// TIA Portal V16 export
// export: Created 2025-11-10T21:24:54.1591457Z, ExportSetting WithDefaults, DisplayName Totally Integrated Automation Portal, DisplayVersion V16, DisplayName TIA Portal Version Control Interface, DisplayVersion V16, DisplayName TIA Portal Openness, DisplayVersion V16, DisplayName STEP 7 Professional, DisplayVersion V16, DisplayName STEP 7 Safety, DisplayVersion V16, DisplayName WinCC Advanced, DisplayVersion V16
ORGANIZATION_BLOCK "OB1"   // OB1, LAD, ProgramCycle
TITLE = MAIN Program - Sweep
VERSION : 0.1
// MAIN Program Block (Release)
// stored: IsIECCheckEnabled false
   VAR_TEMP
      Temp_0 : Byte;
      Temp_1 : Byte;
      Temp_2 : Byte;
      Temp_3 : Byte;
      Temp_4 : Byte;
      Temp_5 : Byte;
      Temp_6 : Int;
      Temp_7 : Int;
      Temp_8 : Int;
      Temp_9 : Date_And_Time;
      Temp_10 : DWord;
      EncoderDirection : Bool;
      HomingActive : Bool;
      EncError : Bool;
      SafetyActive : Bool;
      "Spare Drive 6" : Bool;
      "Spare Drive 7" : Bool;
      "Spare Drive 8" : Bool;
      "Spare Drive 9" : Bool;
      "Spare Drive 10" : Bool;
      SAFE_OK_Signal : Bool;
      Raw_Position : Real;
      Encoder : Int;
      Gate : Bool;
      GATESTP : Bool;
      OTERRA : Bool;
      Direct : Bool;
      Prepar : Bool;
      CMPV1 : Bool;
      CMPV2 : Bool;
      RESSYNC : Bool;
      RESZERO : Bool;
      OTERR : Bool;
      UnscPos : Int;
      Sc_Pos : Int;
      ActEncPos : Real;
      Start_ReferenceRun : Bool;
      ReferenceSwitch_Input : Bool;
      "Reference Position" : Real;
      "Jog FWD" : Bool;
      "Jog REV" : Bool;
      RefSwitchTemp : Bool;
      RefPosDint : DInt;
      RefPosInt : Real;
      Start_Movement : Bool;
      ClockTime : Int;
      LT_Time : Date_And_Time;
      Summer : Bool;
      SystemStartUp : Bool;
      StartupLow : Bool;
      ManualSensorOverride : Bool;
      Axis1_ScaledPosition : Real;
      Axis1_ActualEncPosition : Real;
      ActivateProductBufferV2 : Bool;
      ActivateProductBufferV3 : Bool;
      SetZPulse : Bool;
      Enc2_AboveZero : DInt;
      MinValue : DInt;
      EncBelowZero : Bool;
      SafeEncValue : Real;
      Enc2_Real : Real;
      ScPos : Real;
      UseOldDriveManager : Bool;
      NotUsed : Bool;
      Door2 : Bool;
      Resettt : Bool;
      BlkMovReturn : Int;
      BlkMovReturn2 : Int;
      ServoAxis3RefRun : Bool;
   END_VAR
   VAR_TEMP   // added for the SCL form of the ladder/FBD networks
      _w1 : Bool;
   END_VAR
BEGIN

REGION Network 1: System Startup
   // Network for detecting System Start-up.
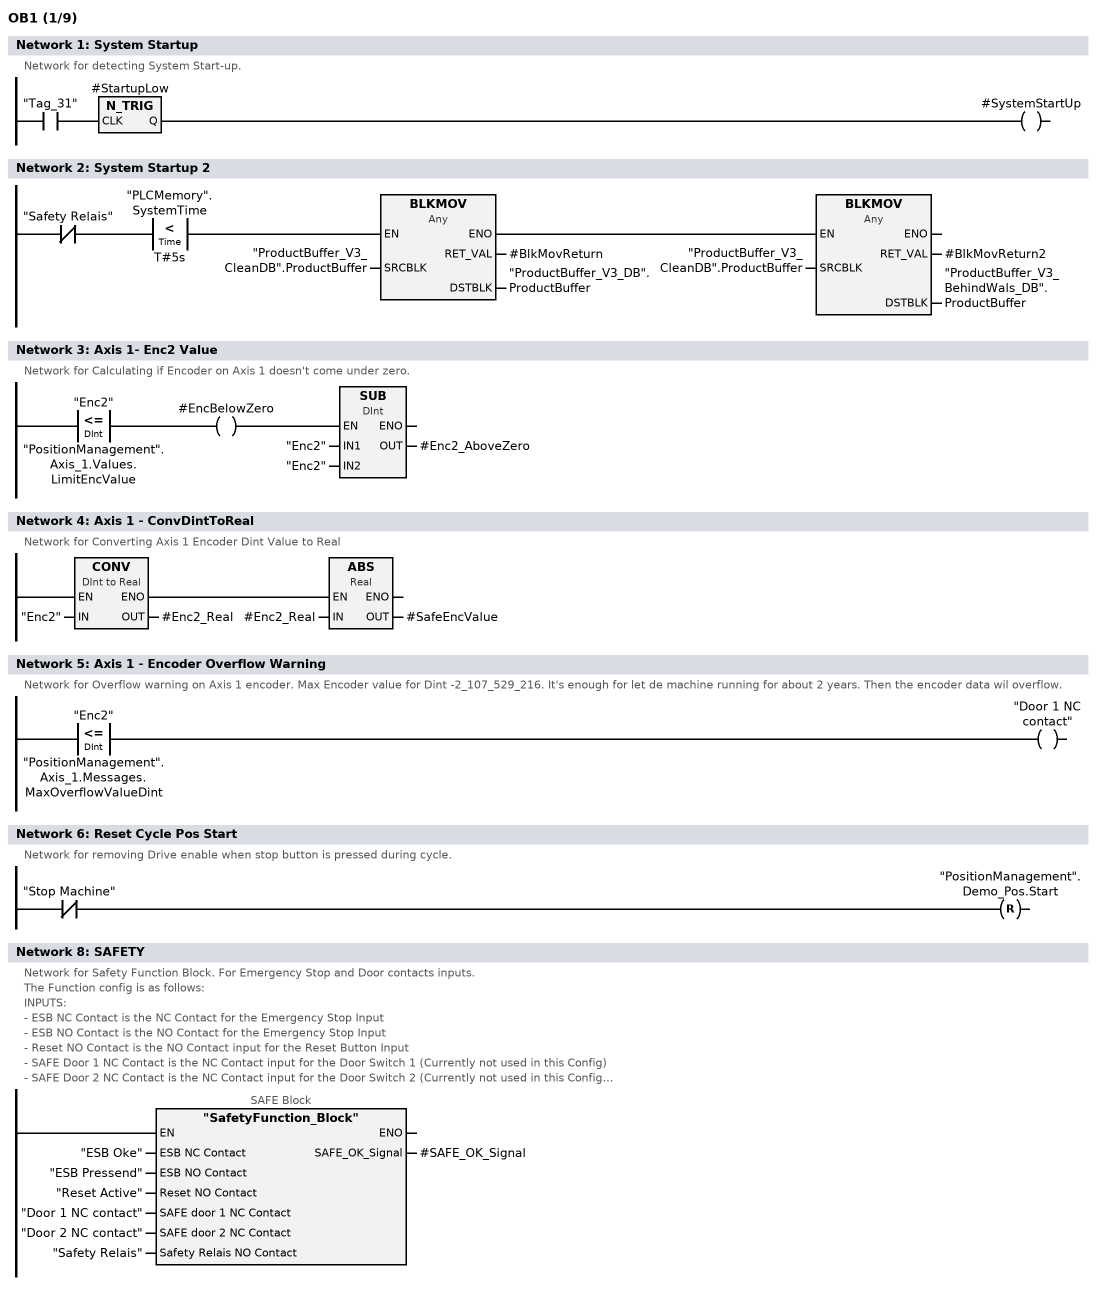
   RUNG wire#powerrail
      Contact( "Tag_31" )
      N_Trig( #StartupLow )
      Coil( #SystemStartUp )
   END_RUNG
   // the same network as SCL:
   #_w1 := NOT "Tag_31" AND #StartupLow;   // falling edge
   #StartupLow := "Tag_31";
   #SystemStartUp := #_w1;
END_REGION

REGION Network 2: System Startup 2
   RUNG wire#powerrail
      I_Contact( "Safety Relais" )
      { S7_Templates := "SrcType := Time" } LT_Contact(in1 := "PLCMemory".SystemTime, in2 := T#5s)
      { S7_Templates := "blk_type := Any" } BLKMOV(SRCBLK := "ProductBuffer_V3_CleanDB".ProductBuffer, RET_VAL => #BlkMovReturn, DSTBLK => "ProductBuffer_V3_DB".ProductBuffer)
      { S7_Templates := "blk_type := Any" } BLKMOV(SRCBLK := "ProductBuffer_V3_CleanDB".ProductBuffer, RET_VAL => #BlkMovReturn2, DSTBLK => "ProductBuffer_V3_BehindWals_DB".ProductBuffer)
   END_RUNG
   // the same network as SCL:
   #BlkMovReturn := BLKMOV(EN := NOT "Safety Relais" AND ("PLCMemory".SystemTime < T#5s),
                           SRCBLK := "ProductBuffer_V3_CleanDB".ProductBuffer,
                           DSTBLK => "ProductBuffer_V3_DB".ProductBuffer,
                           ENO => #_w1);
   IF #_w1 THEN
       #BlkMovReturn2 := BLKMOV(SRCBLK := "ProductBuffer_V3_CleanDB".ProductBuffer,
                               DSTBLK => "ProductBuffer_V3_BehindWals_DB".ProductBuffer);
   END_IF;
END_REGION

REGION Network 3: Axis 1- Enc2 Value
   // Network for Calculating if Encoder on Axis 1 doesn't come under zero.
   RUNG wire#powerrail
      { S7_Templates := "SrcType := DInt" } LE_Contact(in1 := "Enc2", in2 := "PositionManagement".Axis_1.Values.LimitEncValue)
      Coil( #EncBelowZero )
      { S7_Templates := "SrcType := DInt"; S7_GenerateENO := "TRUE" } Sub(in1 := "Enc2", in2 := "Enc2", out => #Enc2_AboveZero)
   END_RUNG
   // the same network as SCL:
   #EncBelowZero := "Enc2" <= "PositionManagement".Axis_1.Values.LimitEncValue;
   IF #EncBelowZero THEN #Enc2_AboveZero := "Enc2" - "Enc2"; END_IF;
END_REGION

REGION Network 4: Axis 1 - ConvDintToReal
   // Network for Converting Axis 1 Encoder Dint Value to Real
   RUNG wire#powerrail
      { S7_Templates := "[SrcType := DInt, DestType := Real]"; S7_GenerateENO := "TRUE" } Convert(in := "Enc2", out => #Enc2_Real)
      { S7_Templates := "SrcType := Real"; S7_GenerateENO := "TRUE" } Abs(in := #Enc2_Real, out => #SafeEncValue)
   END_RUNG
   // the same network as SCL:
   // ENO of a box is taken as its EN; it also drops when the box reports an error
   #Enc2_Real := DINT_TO_REAL("Enc2");
   #SafeEncValue := ABS(#Enc2_Real);
END_REGION

REGION Network 5: Axis 1 - Encoder Overflow Warning
   // Network for Overflow warning on Axis 1 encoder. Max Encoder value for Dint -2_107_529_216. It's enough for let de machine running for about 2 years. Then the encoder data wil overflow.
   RUNG wire#powerrail
      { S7_Templates := "SrcType := DInt" } LE_Contact(in1 := "Enc2", in2 := "PositionManagement".Axis_1.Messages.MaxOverflowValueDint)
      Coil( "Door 1 NC contact" )
   END_RUNG
   // the same network as SCL:
   "Door 1 NC contact" := "Enc2" <= "PositionManagement".Axis_1.Messages.MaxOverflowValueDint;
END_REGION

REGION Network 6: Reset Cycle Pos Start
   // Network for removing Drive enable when stop button is pressed during cycle.
   RUNG wire#powerrail
      I_Contact( "Stop Machine" )
      R_Coil( "PositionManagement".Demo_Pos.Start )
   END_RUNG
   // the same network as SCL:
   IF NOT "Stop Machine" THEN "PositionManagement".Demo_Pos.Start := FALSE; END_IF;
END_REGION

REGION Network 7: Retain Veriables (Not Used)
   // Spare Network Currently not used
END_REGION

REGION Network 8: SAFETY
   // Network for Safety Function Block. For Emergency Stop and Door contacts inputs.
   // The Function config is as follows:
   // 
   // INPUTS:
   // - ESB NC Contact is the NC Contact for the Emergency Stop Input
   // - ESB NO Contact is the NO Contact for the Emergency Stop Input
   // - Reset NO Contact is the NO Contact input for the Reset Button Input
   // - SAFE Door 1 NC Contact is the NC Contact input for the Door Switch 1 (Currently not used in this Config)
   // - SAFE Door 2 NC Contact is the NC Contact input for the Door Switch 2 (Currently not used in this Config)
   // - Safety Relais NO Contact is the NO Contact Input for feedback whenether the Safety Relais is powered or not.
   // 
   // OUTPUTS:
   // - SAFE_OK_Signal is the output for the SAFE OK signal, it's HIGH when all safety inputs are HIGH, en when Reset is given.
   RUNG wire#powerrail
      "SafetyFunction_Block"("ESB NC Contact" := "ESB Oke", "ESB NO Contact" := "ESB Pressend", "Reset NO Contact" := "Reset Active", "SAFE door 1 NC Contact" := "Door 1 NC contact", "SAFE door 2 NC Contact" := "Door 2 NC contact", "Safety Relais NO Contact" := "Safety Relais", SAFE_OK_Signal => #SAFE_OK_Signal)   // SAFE Block
   END_RUNG
   // the same network as SCL:
   "SafetyFunction_Block"("ESB NC Contact" := "ESB Oke",   // SAFE Block
                          "ESB NO Contact" := "ESB Pressend",
                          "Reset NO Contact" := "Reset Active",
                          "SAFE door 1 NC Contact" := "Door 1 NC contact",
                          "SAFE door 2 NC Contact" := "Door 2 NC contact",
                          "Safety Relais NO Contact" := "Safety Relais",
                          SAFE_OK_Signal => #SAFE_OK_Signal);
END_REGION

REGION Network 9: SAFE Signal
   // Network for internal SAFETY OK Confirmation
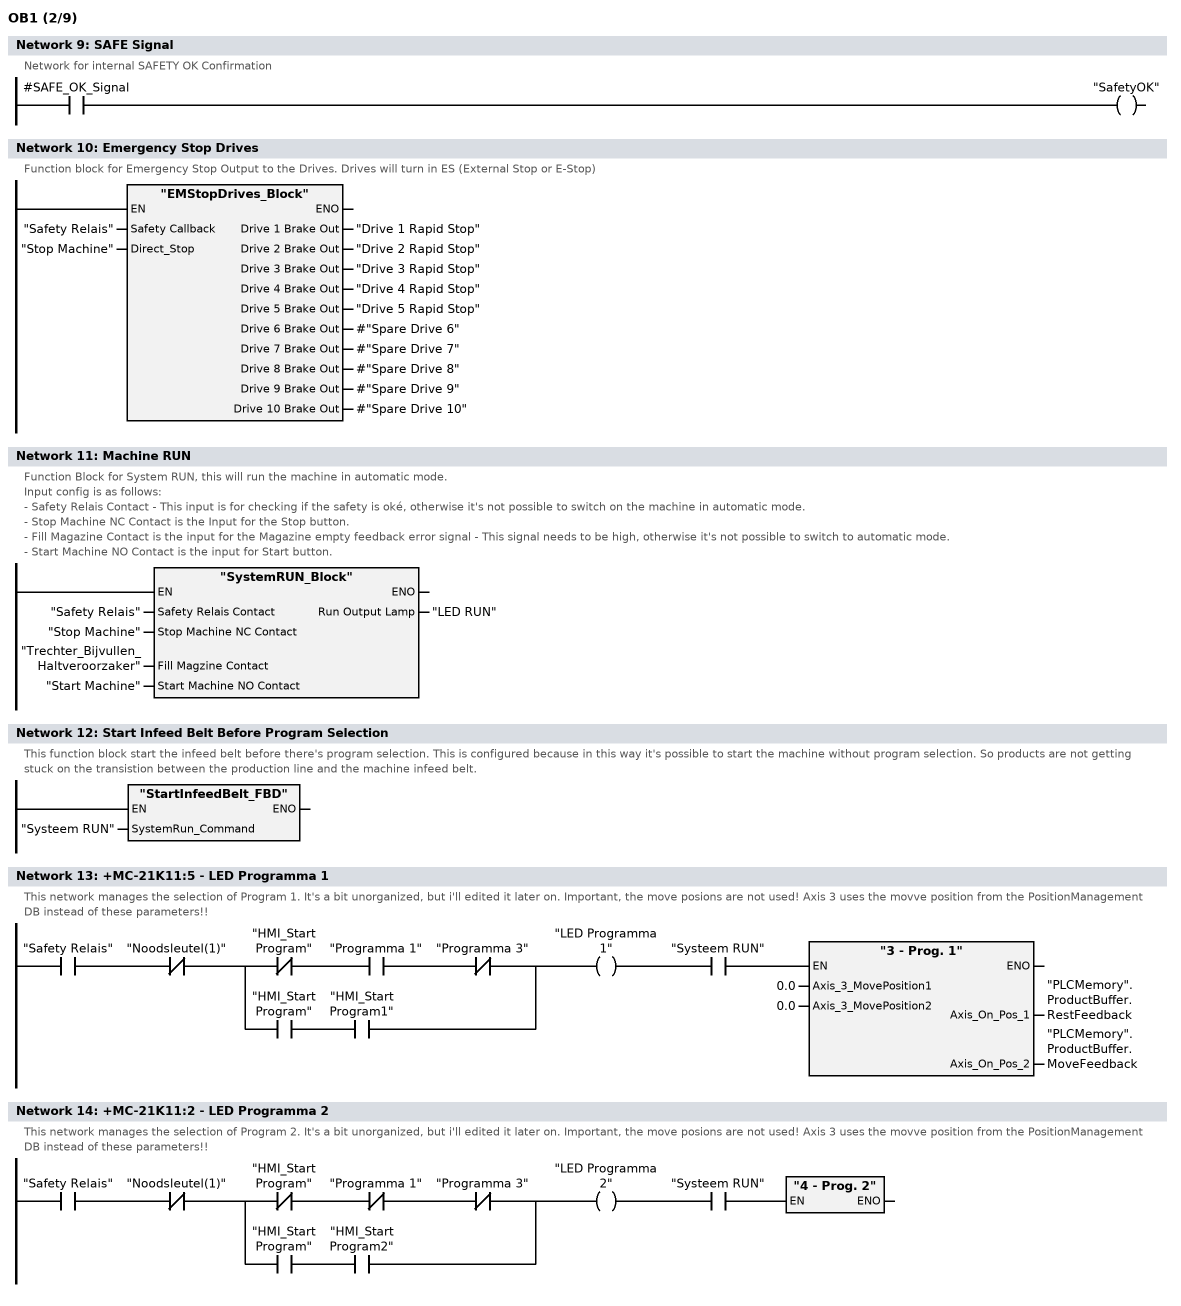
   RUNG wire#powerrail
      Contact( #SAFE_OK_Signal )
      Coil( "SafetyOK" )
   END_RUNG
   // the same network as SCL:
   "SafetyOK" := #SAFE_OK_Signal;
END_REGION

REGION Network 10: Emergency Stop Drives
   // Function block for Emergency Stop Output to the Drives. Drives will turn in ES (External Stop or E-Stop)
   RUNG wire#powerrail
      "EMStopDrives_Block"("Safety Callback" := "Safety Relais", Direct_Stop := "Stop Machine", "Drive 1 Brake Out" => "Drive 1 Rapid Stop", "Drive 2 Brake Out" => "Drive 2 Rapid Stop", "Drive 3 Brake Out" => "Drive 3 Rapid Stop", "Drive 4 Brake Out" => "Drive 4 Rapid Stop", "Drive 5 Brake Out" => "Drive 5 Rapid Stop", "Drive 6 Brake Out" => #"Spare Drive 6", "Drive 7 Brake Out" => #"Spare Drive 7", "Drive 8 Brake Out" => #"Spare Drive 8", "Drive 9 Brake Out" => #"Spare Drive 9", "Drive 10 Brake Out" => #"Spare Drive 10")
   END_RUNG
   // the same network as SCL:
   "EMStopDrives_Block"("Safety Callback" := "Safety Relais",
                        Direct_Stop := "Stop Machine",
                        "Drive 1 Brake Out" => "Drive 1 Rapid Stop",
                        "Drive 2 Brake Out" => "Drive 2 Rapid Stop",
                        "Drive 3 Brake Out" => "Drive 3 Rapid Stop",
                        "Drive 4 Brake Out" => "Drive 4 Rapid Stop",
                        "Drive 5 Brake Out" => "Drive 5 Rapid Stop",
                        "Drive 6 Brake Out" => #"Spare Drive 6",
                        "Drive 7 Brake Out" => #"Spare Drive 7",
                        "Drive 8 Brake Out" => #"Spare Drive 8",
                        "Drive 9 Brake Out" => #"Spare Drive 9",
                        "Drive 10 Brake Out" => #"Spare Drive 10");
END_REGION

REGION Network 11: Machine RUN
   // Function Block for System RUN, this will run the machine in automatic mode.
   // Input config is as follows:
   // - Safety Relais Contact - This input is for checking if the safety is oké, otherwise it's not possible to switch on the machine in automatic mode.
   // - Stop Machine NC Contact is the Input for the Stop button.
   // - Fill Magazine Contact is the input for the Magazine empty feedback error signal - This signal needs to be high, otherwise it's not possible to switch to automatic mode.
   // - Start Machine NO Contact is the input for Start button.
   RUNG wire#powerrail
      "SystemRUN_Block"("Safety Relais Contact" := "Safety Relais", "Stop Machine NC Contact" := "Stop Machine", "Fill Magzine Contact" := "Trechter_Bijvullen_Haltveroorzaker", "Start Machine NO Contact" := "Start Machine", "Run Output Lamp" => "LED RUN")
   END_RUNG
   // the same network as SCL:
   "SystemRUN_Block"("Safety Relais Contact" := "Safety Relais",
                     "Stop Machine NC Contact" := "Stop Machine",
                     "Fill Magzine Contact" := "Trechter_Bijvullen_Haltveroorzaker",
                     "Start Machine NO Contact" := "Start Machine",
                     "Run Output Lamp" => "LED RUN");
END_REGION

REGION Network 12: Start Infeed Belt Before Program Selection
   // This function block start the infeed belt before there's program selection. This is configured because in this way it's possible to start the machine without program selection. So products are not getting stuck on the transistion between the production line and the machine infeed belt.
   RUNG wire#powerrail
      "StartInfeedBelt_FBD"(SystemRun_Command := "Systeem RUN")
   END_RUNG
   // the same network as SCL:
   "StartInfeedBelt_FBD"(SystemRun_Command := "Systeem RUN");
END_REGION

REGION Network 13: +MC-21K11:5 - LED Programma 1
   // This network manages the selection of Program 1. It's a bit unorganized, but i'll edited it later on. Important, the move posions are not used! Axis 3 uses the movve position from the PositionManagement DB instead of these parameters!!
   RUNG wire#powerrail
      Contact( "Safety Relais" )
      I_Contact( "Noodsleutel(1)" )
      wire#w1
      I_Contact( "HMI_StartProgram" )
      Contact( "Programma 1" )
      I_Contact( "Programma 3" )
      wire#w2
      Coil( "LED Programma 1" )
      Contact( "Systeem RUN" )
      "3 - Prog. 1"(Axis_3_MovePosition1 := 0.0, Axis_3_MovePosition2 := 0.0, Axis_On_Pos_1 => "PLCMemory".ProductBuffer.RestFeedback, Axis_On_Pos_2 => "PLCMemory".ProductBuffer.MoveFeedback)
   END_RUNG
   RUNG wire#w1
      Contact( "HMI_StartProgram" )
      Contact( "HMI_StartProgram1" )
   END_RUNG wire#w2
   // the same network as SCL:
   "LED Programma 1" := "Safety Relais" AND NOT "Noodsleutel(1)" AND ((NOT "HMI_StartProgram" AND "Programma 1" AND NOT "Programma 3") OR ("HMI_StartProgram" AND "HMI_StartProgram1"));
   IF "LED Programma 1" AND "Systeem RUN" THEN
       "3 - Prog. 1"(Axis_3_MovePosition1 := 0.0,
                     Axis_3_MovePosition2 := 0.0,
                     Axis_On_Pos_1 => "PLCMemory".ProductBuffer.RestFeedback,
                     Axis_On_Pos_2 => "PLCMemory".ProductBuffer.MoveFeedback);
   END_IF;
END_REGION

REGION Network 14: +MC-21K11:2 - LED Programma 2
   // This network manages the selection of Program 2. It's a bit unorganized, but i'll edited it later on. Important, the move posions are not used! Axis 3 uses the movve position from the PositionManagement DB instead of these parameters!!
   RUNG wire#powerrail
      Contact( "Safety Relais" )
      I_Contact( "Noodsleutel(1)" )
      wire#w1
      I_Contact( "HMI_StartProgram" )
      I_Contact( "Programma 1" )
      I_Contact( "Programma 3" )
      wire#w2
      Coil( "LED Programma 2" )
      Contact( "Systeem RUN" )
      "4 - Prog. 2"()
   END_RUNG
   RUNG wire#w1
      Contact( "HMI_StartProgram" )
      Contact( "HMI_StartProgram2" )
   END_RUNG wire#w2
   // the same network as SCL:
   "LED Programma 2" := "Safety Relais" AND NOT "Noodsleutel(1)" AND ((NOT "HMI_StartProgram" AND NOT "Programma 1" AND NOT "Programma 3") OR ("HMI_StartProgram" AND "HMI_StartProgram2"));
   IF "LED Programma 2" AND "Systeem RUN" THEN "4 - Prog. 2"(); END_IF;
END_REGION

REGION Network 15: +MC-21K11:6 - LED Programma 3
   // This network manages the selection of Program 3. It's a bit unorganized, but i'll edited it later on. Important, the move posions are not used! Axis 3 uses the movve position from the PositionManagement DB instead of these parameters!!
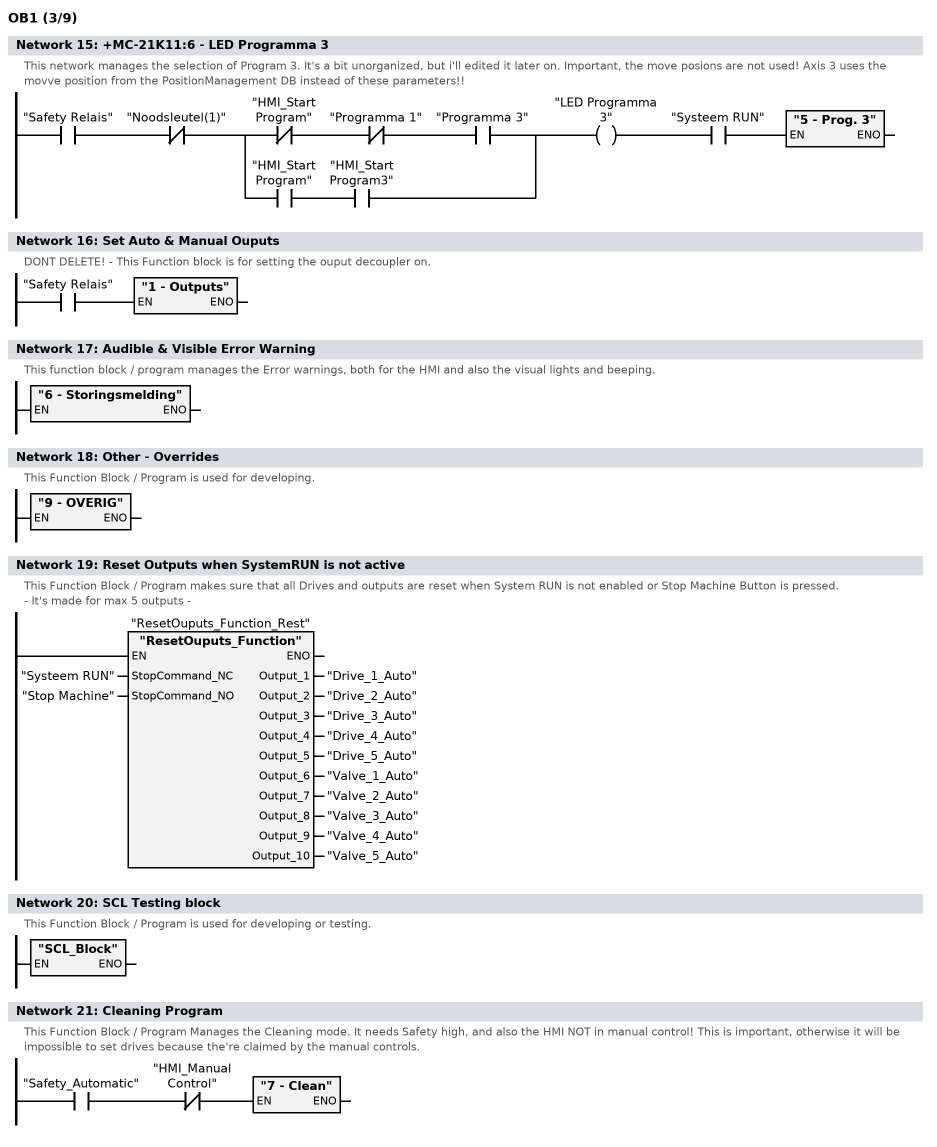
   RUNG wire#powerrail
      Contact( "Safety Relais" )
      I_Contact( "Noodsleutel(1)" )
      wire#w1
      I_Contact( "HMI_StartProgram" )
      I_Contact( "Programma 1" )
      Contact( "Programma 3" )
      wire#w2
      Coil( "LED Programma 3" )
      Contact( "Systeem RUN" )
      "5 - Prog. 3"()
   END_RUNG
   RUNG wire#w1
      Contact( "HMI_StartProgram" )
      Contact( "HMI_StartProgram3" )
   END_RUNG wire#w2
   // the same network as SCL:
   "LED Programma 3" := "Safety Relais" AND NOT "Noodsleutel(1)" AND ((NOT "HMI_StartProgram" AND NOT "Programma 1" AND "Programma 3") OR ("HMI_StartProgram" AND "HMI_StartProgram3"));
   IF "LED Programma 3" AND "Systeem RUN" THEN "5 - Prog. 3"(); END_IF;
END_REGION

REGION Network 16: Set Auto & Manual Ouputs
   // DONT DELETE! - This Function block is for setting the ouput decoupler on.
   RUNG wire#powerrail
      Contact( "Safety Relais" )
      "1 - Outputs"()
   END_RUNG
   // the same network as SCL:
   IF "Safety Relais" THEN "1 - Outputs"(); END_IF;
END_REGION

REGION Network 17: Audible & Visible Error Warning
   // This function block / program manages the Error warnings, both for the HMI and also the visual lights and beeping.
   RUNG wire#powerrail
      "6 - Storingsmelding"()
   END_RUNG
   // the same network as SCL:
   "6 - Storingsmelding"();
END_REGION

REGION Network 18: Other - Overrides
   // This Function Block / Program is used for developing.
   RUNG wire#powerrail
      "9 - OVERIG"()
   END_RUNG
   // the same network as SCL:
   "9 - OVERIG"();
END_REGION

REGION Network 19: Reset Outputs when SystemRUN is not active
   // This Function Block / Program makes sure that all Drives and outputs are reset when System RUN is not enabled or Stop Machine Button is pressed. 
   // - It's made for max 5 outputs -
   RUNG wire#powerrail
      "ResetOuputs_Function_Rest"(StopCommand_NC := "Systeem RUN", StopCommand_NO := "Stop Machine", Output_1 => "Drive_1_Auto", Output_2 => "Drive_2_Auto", Output_3 => "Drive_3_Auto", Output_4 => "Drive_4_Auto", Output_5 => "Drive_5_Auto", Output_6 => "Valve_1_Auto", Output_7 => "Valve_2_Auto", Output_8 => "Valve_3_Auto", Output_9 => "Valve_4_Auto", Output_10 => "Valve_5_Auto")
   END_RUNG
   // the same network as SCL:
   "ResetOuputs_Function_Rest"(StopCommand_NC := "Systeem RUN",   // "ResetOuputs_Function"
                           StopCommand_NO := "Stop Machine",
                           Output_1 => "Drive_1_Auto",
                           Output_2 => "Drive_2_Auto",
                           Output_3 => "Drive_3_Auto",
                           Output_4 => "Drive_4_Auto",
                           Output_5 => "Drive_5_Auto",
                           Output_6 => "Valve_1_Auto",
                           Output_7 => "Valve_2_Auto",
                           Output_8 => "Valve_3_Auto",
                           Output_9 => "Valve_4_Auto",
                           Output_10 => "Valve_5_Auto");
END_REGION

REGION Network 20: SCL Testing block
   // This Function Block / Program is used for developing or testing.
   RUNG wire#powerrail
      "SCL_Block"()
   END_RUNG
   // the same network as SCL:
   "SCL_Block"();
END_REGION

REGION Network 21: Cleaning Program
   // This Function Block / Program Manages the Cleaning mode. It needs Safety high, and also the HMI NOT in manual control! This is important, otherwise it will be impossible to set drives because the're claimed by the manual controls.
   RUNG wire#powerrail
      Contact( "Safety_Automatic" )
      I_Contact( "HMI_ManualControl" )
      "7 - Clean"()
   END_RUNG
   // the same network as SCL:
   IF "Safety_Automatic" AND NOT "HMI_ManualControl" THEN "7 - Clean"(); END_IF;
END_REGION

REGION Network 22: Ref Switch Axis 3 - Delay Ref Switch
   // This short code helps putting a short filter on Sensor of Axis 3.
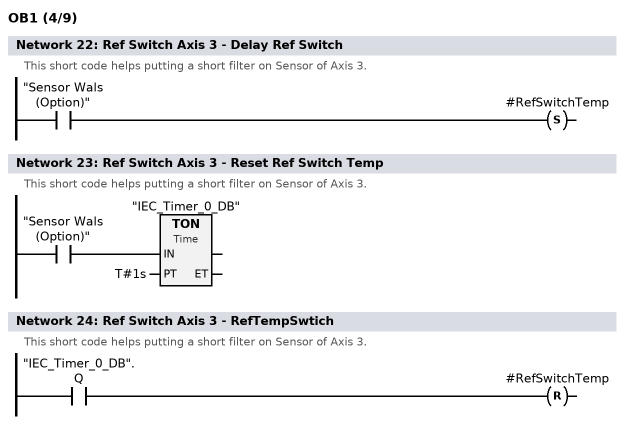
   RUNG wire#powerrail
      Contact( "Sensor Wals (Option)" )
      S_Coil( #RefSwitchTemp )
   END_RUNG
   // the same network as SCL:
   IF "Sensor Wals (Option)" THEN #RefSwitchTemp := TRUE; END_IF;
END_REGION

REGION Network 23: Ref Switch Axis 3 - Reset Ref Switch Temp
   // This short code helps putting a short filter on Sensor of Axis 3.
   RUNG wire#powerrail
      Contact( "Sensor Wals (Option)" )
      { S7_Templates := "time_type := Time" } "IEC_Timer_0_DB".TON(pt := T#1s, et =>)
   END_RUNG
   // the same network as SCL:
   "IEC_Timer_0_DB".TON(IN := "Sensor Wals (Option)", PT := T#1s);
END_REGION

REGION Network 24: Ref Switch Axis 3 - RefTempSwtich
   // This short code helps putting a short filter on Sensor of Axis 3.
   RUNG wire#powerrail
      Contact( "IEC_Timer_0_DB".Q )
      R_Coil( #RefSwitchTemp )
   END_RUNG
   // the same network as SCL:
   IF "IEC_Timer_0_DB".Q THEN #RefSwitchTemp := FALSE; END_IF;
END_REGION

REGION Network 25: Drive Manager Axis 3
   // This is the Drive Manager function block, it controls the Asynchronous Servo Axis combined with an Siko IG06 Encoder. More about this can be found on the wiki page on Notion.
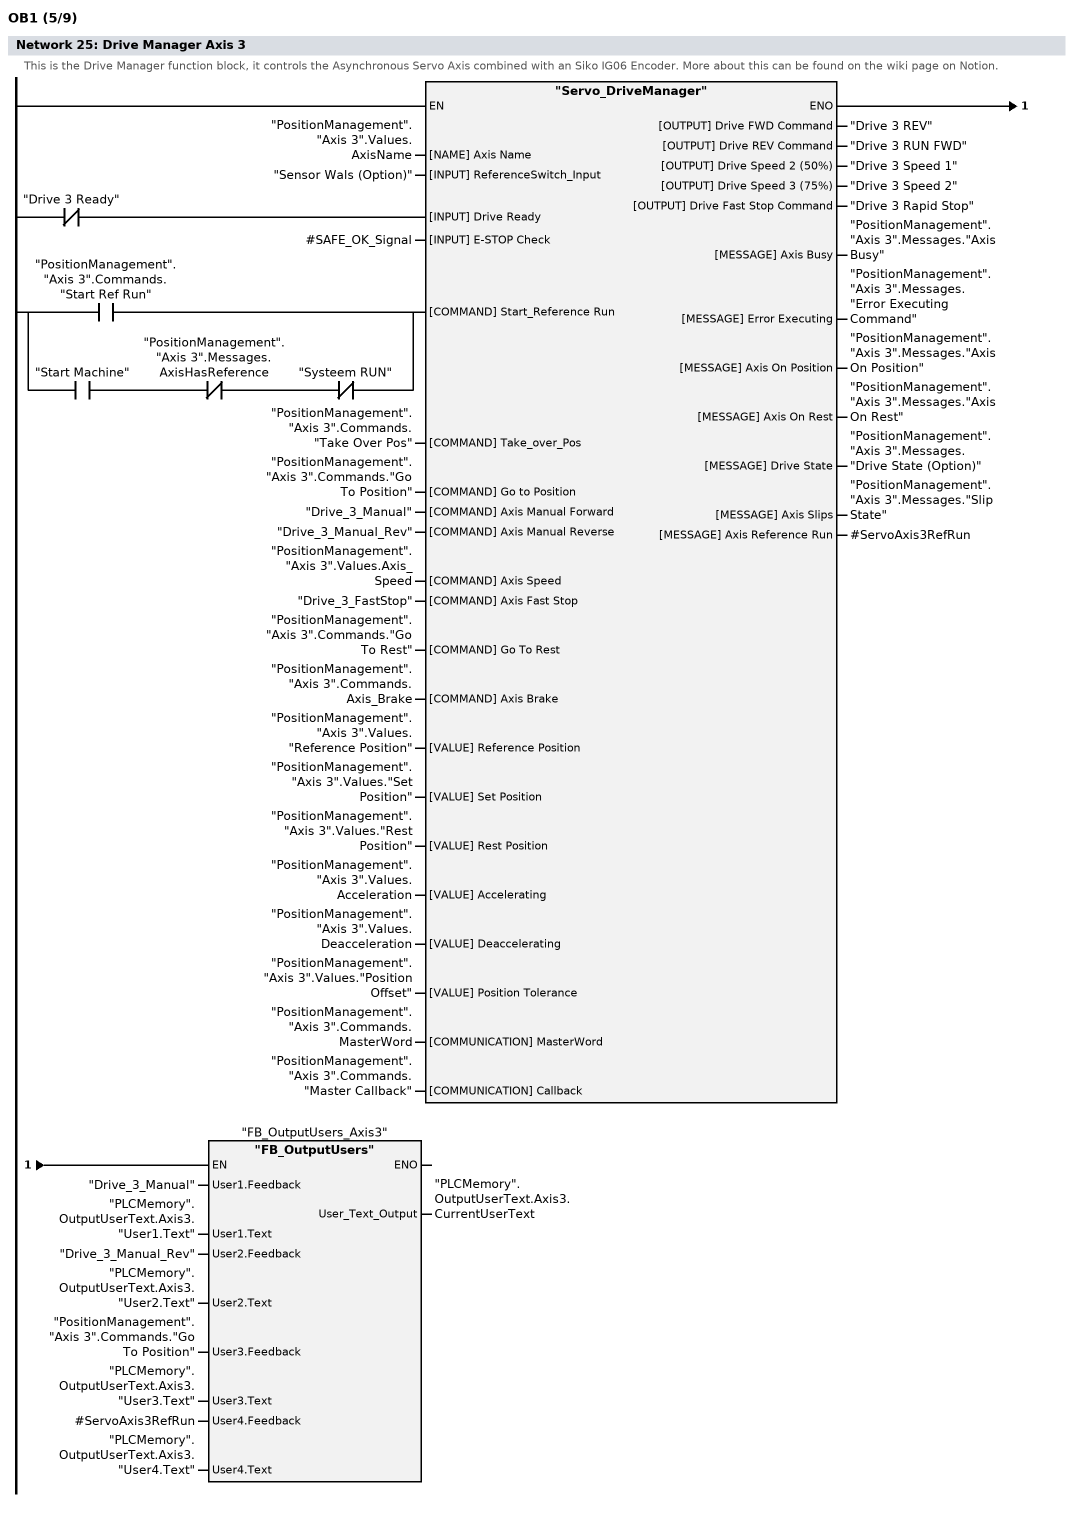
   RUNG wire#powerrail
      "Servo_DriveManager"("[INPUT] Drive Ready" := wire#w1, "[COMMAND] Start_Reference Run" := wire#w2, "[NAME] Axis Name" := "PositionManagement"."Axis 3".Values.AxisName, "[INPUT] ReferenceSwitch_Input" := "Sensor Wals (Option)", "[INPUT] E-STOP Check" := #SAFE_OK_Signal, "[COMMAND] Take_over_Pos" := "PositionManagement"."Axis 3".Commands."Take Over Pos", "[COMMAND] Go to Position" := "PositionManagement"."Axis 3".Commands."Go To Position", "[COMMAND] Axis Manual Forward" := "Drive_3_Manual", "[COMMAND] Axis Manual Reverse" := "Drive_3_Manual_Rev", "[COMMAND] Axis Speed" := "PositionManagement"."Axis 3".Values.Axis_Speed, "[COMMAND] Axis Fast Stop" := "Drive_3_FastStop", "[COMMAND] Go To Rest" := "PositionManagement"."Axis 3".Commands."Go To Rest", "[COMMAND] Axis Brake" := "PositionManagement"."Axis 3".Commands.Axis_Brake, "[VALUE] Reference Position" := "PositionManagement"."Axis 3".Values."Reference Position", "[VALUE] Set Position" := "PositionManagement"."Axis 3".Values."Set Position", "[VALUE] Rest Position" := "PositionManagement"."Axis 3".Values."Rest Position", "[VALUE] Accelerating" := "PositionManagement"."Axis 3".Values.Acceleration, "[VALUE] Deaccelerating" := "PositionManagement"."Axis 3".Values.Deacceleration, "[VALUE] Position Tolerance" := "PositionManagement"."Axis 3".Values."Position Offset", "[COMMUNICATION] MasterWord" := "PositionManagement"."Axis 3".Commands.MasterWord, "[COMMUNICATION] Callback" := "PositionManagement"."Axis 3".Commands."Master Callback", "[OUTPUT] Drive FWD Command" => "Drive 3 REV", "[OUTPUT] Drive REV Command" => "Drive 3 RUN FWD", "[OUTPUT] Drive Speed 2 (50%)" => "Drive 3 Speed 1", "[OUTPUT] Drive Speed 3 (75%)" => "Drive 3 Speed 2", "[OUTPUT] Drive Fast Stop Command" => "Drive 3 Rapid Stop", "[MESSAGE] Axis Busy" => "PositionManagement"."Axis 3".Messages."Axis Busy", "[MESSAGE] Error Executing" => "PositionManagement"."Axis 3".Messages."Error Executing Command", "[MESSAGE] Axis On Position" => "PositionManagement"."Axis 3".Messages."Axis On Position", "[MESSAGE] Axis On Rest" => "PositionManagement"."Axis 3".Messages."Axis On Rest", "[MESSAGE] Drive State" => "PositionManagement"."Axis 3".Messages."Drive State (Option)", "[MESSAGE] Axis Slips" => "PositionManagement"."Axis 3".Messages."Slip State", "[MESSAGE] Axis Reference Run" => #ServoAxis3RefRun)
      "FB_OutputUsers_Axis3"("User1.Feedback" := "Drive_3_Manual", "User1.Text" := "PLCMemory".OutputUserText.Axis3."User1.Text", "User2.Feedback" := "Drive_3_Manual_Rev", "User2.Text" := "PLCMemory".OutputUserText.Axis3."User2.Text", "User3.Feedback" := "PositionManagement"."Axis 3".Commands."Go To Position", "User3.Text" := "PLCMemory".OutputUserText.Axis3."User3.Text", "User4.Feedback" := #ServoAxis3RefRun, "User4.Text" := "PLCMemory".OutputUserText.Axis3."User4.Text", User_Text_Output => "PLCMemory".OutputUserText.Axis3.CurrentUserText)
   END_RUNG
   RUNG wire#powerrail
      I_Contact( "Drive 3 Ready" )
   END_RUNG wire#w1
   RUNG wire#powerrail
      Contact( "PositionManagement"."Axis 3".Commands."Start Ref Run" )
   END_RUNG wire#w2
   RUNG wire#powerrail
      Contact( "Start Machine" )
      I_Contact( "PositionManagement"."Axis 3".Messages.AxisHasReference )
      I_Contact( "Systeem RUN" )
   END_RUNG wire#w2
   // the same network as SCL:
   "Servo_DriveManager"("[NAME] Axis Name" := "PositionManagement"."Axis 3".Values.AxisName,
                        "[INPUT] ReferenceSwitch_Input" := "Sensor Wals (Option)",
                        "[INPUT] Drive Ready" := NOT "Drive 3 Ready",
                        "[INPUT] E-STOP Check" := #SAFE_OK_Signal,
                        "[COMMAND] Start_Reference Run" := "PositionManagement"."Axis 3".Commands."Start Ref Run" OR ("Start Machine" AND NOT "PositionManagement"."Axis 3".Messages.AxisHasReference AND NOT "Systeem RUN"),
                        "[COMMAND] Take_over_Pos" := "PositionManagement"."Axis 3".Commands."Take Over Pos",
                        "[COMMAND] Go to Position" := "PositionManagement"."Axis 3".Commands."Go To Position",
                        "[COMMAND] Axis Manual Forward" := "Drive_3_Manual",
                        "[COMMAND] Axis Manual Reverse" := "Drive_3_Manual_Rev",
                        "[COMMAND] Axis Speed" := "PositionManagement"."Axis 3".Values.Axis_Speed,
                        "[COMMAND] Axis Fast Stop" := "Drive_3_FastStop",
                        "[COMMAND] Go To Rest" := "PositionManagement"."Axis 3".Commands."Go To Rest",
                        "[COMMAND] Axis Brake" := "PositionManagement"."Axis 3".Commands.Axis_Brake,
                        "[VALUE] Reference Position" := "PositionManagement"."Axis 3".Values."Reference Position",
                        "[VALUE] Set Position" := "PositionManagement"."Axis 3".Values."Set Position",
                        "[VALUE] Rest Position" := "PositionManagement"."Axis 3".Values."Rest Position",
                        "[VALUE] Accelerating" := "PositionManagement"."Axis 3".Values.Acceleration,
                        "[VALUE] Deaccelerating" := "PositionManagement"."Axis 3".Values.Deacceleration,
                        "[VALUE] Position Tolerance" := "PositionManagement"."Axis 3".Values."Position Offset",
                        "[COMMUNICATION] MasterWord" := "PositionManagement"."Axis 3".Commands.MasterWord,
                        "[COMMUNICATION] Callback" := "PositionManagement"."Axis 3".Commands."Master Callback",
                        "[OUTPUT] Drive FWD Command" => "Drive 3 REV",
                        "[OUTPUT] Drive REV Command" => "Drive 3 RUN FWD",
                        "[OUTPUT] Drive Speed 2 (50%)" => "Drive 3 Speed 1",
                        "[OUTPUT] Drive Speed 3 (75%)" => "Drive 3 Speed 2",
                        "[OUTPUT] Drive Fast Stop Command" => "Drive 3 Rapid Stop",
                        "[MESSAGE] Axis Busy" => "PositionManagement"."Axis 3".Messages."Axis Busy",
                        "[MESSAGE] Error Executing" => "PositionManagement"."Axis 3".Messages."Error Executing Command",
                        "[MESSAGE] Axis On Position" => "PositionManagement"."Axis 3".Messages."Axis On Position",
                        "[MESSAGE] Axis On Rest" => "PositionManagement"."Axis 3".Messages."Axis On Rest",
                        "[MESSAGE] Drive State" => "PositionManagement"."Axis 3".Messages."Drive State (Option)",
                        "[MESSAGE] Axis Slips" => "PositionManagement"."Axis 3".Messages."Slip State",
                        "[MESSAGE] Axis Reference Run" => #ServoAxis3RefRun,
                        ENO => #_w1);
   IF #_w1 THEN
       "FB_OutputUsers_Axis3"("User1.Feedback" := "Drive_3_Manual",   // "FB_OutputUsers"
                              "User1.Text" := "PLCMemory".OutputUserText.Axis3."User1.Text",
                              "User2.Feedback" := "Drive_3_Manual_Rev",
                              "User2.Text" := "PLCMemory".OutputUserText.Axis3."User2.Text",
                              "User3.Feedback" := "PositionManagement"."Axis 3".Commands."Go To Position",
                              "User3.Text" := "PLCMemory".OutputUserText.Axis3."User3.Text",
                              "User4.Feedback" := #ServoAxis3RefRun,
                              "User4.Text" := "PLCMemory".OutputUserText.Axis3."User4.Text",
                              User_Text_Output => "PLCMemory".OutputUserText.Axis3.CurrentUserText);
   END_IF;
END_REGION

REGION Network 26: Noodsleutel
   // This Function Block/ Program is for the use of the Noodsleutel, when this input is HIGH, the infeed conveyorbelt is only turning.
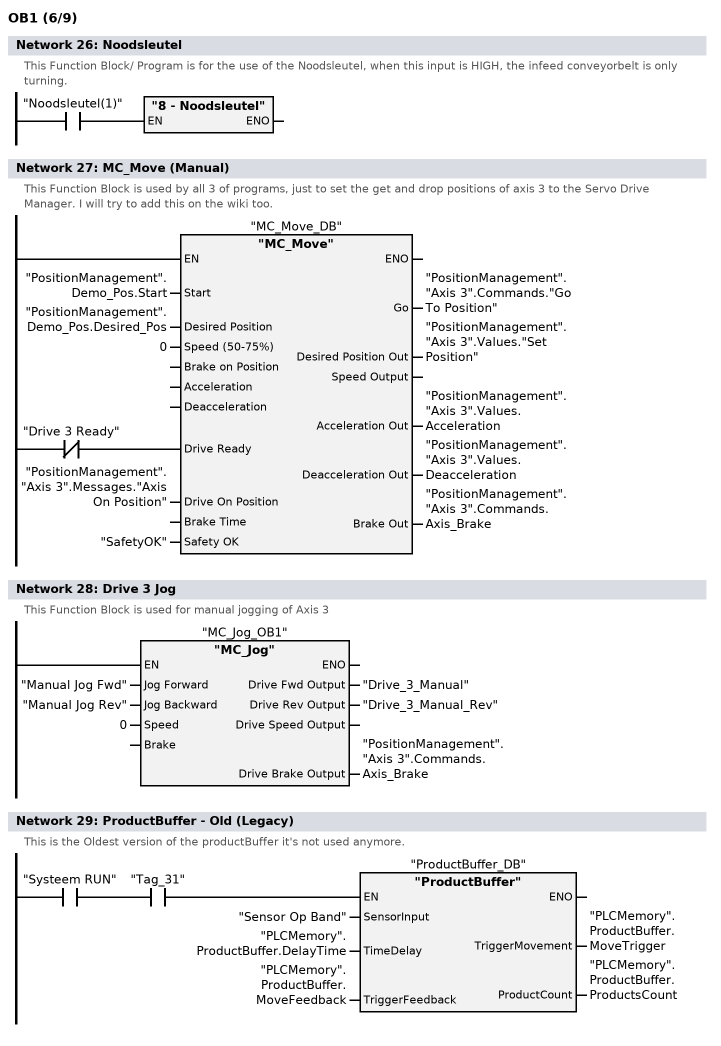
   RUNG wire#powerrail
      Contact( "Noodsleutel(1)" )
      "8 - Noodsleutel"()
   END_RUNG
   // the same network as SCL:
   IF "Noodsleutel(1)" THEN "8 - Noodsleutel"(); END_IF;
END_REGION

REGION Network 27: MC_Move (Manual)
   // This Function Block is used by all 3 of programs, just to set the get and drop positions of axis 3 to the Servo Drive Manager. I will try to add this on the wiki too.
   RUNG wire#powerrail
      "MC_Move_DB"("Drive Ready" := wire#w1, Start := "PositionManagement".Demo_Pos.Start, "Desired Position" := "PositionManagement".Demo_Pos.Desired_Pos, "Speed (50-75%)" := 0, "Brake on Position" :=, Acceleration :=, Deacceleration :=, "Drive On Position" := "PositionManagement"."Axis 3".Messages."Axis On Position", "Brake Time" :=, "Safety OK" := "SafetyOK", Go => "PositionManagement"."Axis 3".Commands."Go To Position", "Desired Position Out" => "PositionManagement"."Axis 3".Values."Set Position", "Speed Output" =>, "Acceleration Out" => "PositionManagement"."Axis 3".Values.Acceleration, "Deacceleration Out" => "PositionManagement"."Axis 3".Values.Deacceleration, "Brake Out" => "PositionManagement"."Axis 3".Commands.Axis_Brake)
   END_RUNG
   RUNG wire#powerrail
      I_Contact( "Drive 3 Ready" )
   END_RUNG wire#w1
   // the same network as SCL:
   "MC_Move_DB"(Start := "PositionManagement".Demo_Pos.Start,   // "MC_Move"
                "Desired Position" := "PositionManagement".Demo_Pos.Desired_Pos,
                "Speed (50-75%)" := 0,
                "Drive Ready" := NOT "Drive 3 Ready",
                "Drive On Position" := "PositionManagement"."Axis 3".Messages."Axis On Position",
                "Safety OK" := "SafetyOK",
                Go => "PositionManagement"."Axis 3".Commands."Go To Position",
                "Desired Position Out" => "PositionManagement"."Axis 3".Values."Set Position",
                "Acceleration Out" => "PositionManagement"."Axis 3".Values.Acceleration,
                "Deacceleration Out" => "PositionManagement"."Axis 3".Values.Deacceleration,
                "Brake Out" => "PositionManagement"."Axis 3".Commands.Axis_Brake);
END_REGION

REGION Network 28: Drive 3 Jog
   // This Function Block is used for manual jogging of Axis 3
   RUNG wire#powerrail
      "MC_Jog_OB1"("Jog Forward" := "Manual Jog Fwd", "Jog Backward" := "Manual Jog Rev", Speed := 0, Brake :=, "Drive Fwd Output" => "Drive_3_Manual", "Drive Rev Output" => "Drive_3_Manual_Rev", "Drive Speed Output" =>, "Drive Brake Output" => "PositionManagement"."Axis 3".Commands.Axis_Brake)
   END_RUNG
   // the same network as SCL:
   "MC_Jog_OB1"("Jog Forward" := "Manual Jog Fwd",   // "MC_Jog"
                "Jog Backward" := "Manual Jog Rev",
                Speed := 0,
                "Drive Fwd Output" => "Drive_3_Manual",
                "Drive Rev Output" => "Drive_3_Manual_Rev",
                "Drive Brake Output" => "PositionManagement"."Axis 3".Commands.Axis_Brake);
END_REGION

REGION Network 29: ProductBuffer - Old (Legacy)
   // This is the Oldest version of the productBuffer it's not used anymore.
   RUNG wire#powerrail
      Contact( "Systeem RUN" )
      Contact( "Tag_31" )
      "ProductBuffer_DB"(SensorInput := "Sensor Op Band", TimeDelay := "PLCMemory".ProductBuffer.DelayTime, TriggerFeedback := "PLCMemory".ProductBuffer.MoveFeedback, TriggerMovement => "PLCMemory".ProductBuffer.MoveTrigger, ProductCount => "PLCMemory".ProductBuffer.ProductsCount)
   END_RUNG
   // the same network as SCL:
   IF "Systeem RUN" AND "Tag_31" THEN
       "ProductBuffer_DB"(SensorInput := "Sensor Op Band",   // "ProductBuffer"
                          TimeDelay := "PLCMemory".ProductBuffer.DelayTime,
                          TriggerFeedback := "PLCMemory".ProductBuffer.MoveFeedback,
                          TriggerMovement => "PLCMemory".ProductBuffer.MoveTrigger,
                          ProductCount => "PLCMemory".ProductBuffer.ProductsCount);
   END_IF;
END_REGION

REGION Network 30: ProductBuffer V2 (Old - Don't use!)
   // This is Version 2 of the product buffer, and also not used anymore.
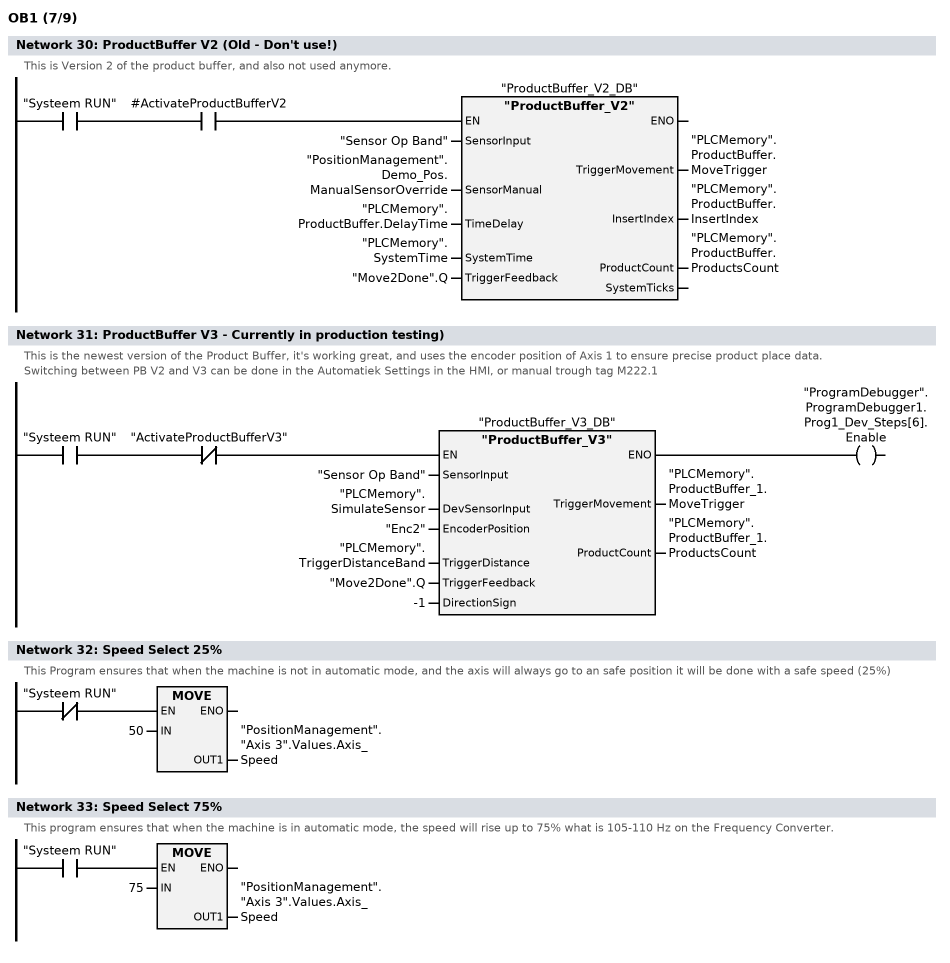
   RUNG wire#powerrail
      Contact( "Systeem RUN" )
      Contact( #ActivateProductBufferV2 )
      "ProductBuffer_V2_DB"(SensorInput := "Sensor Op Band", SensorManual := "PositionManagement".Demo_Pos.ManualSensorOverride, TimeDelay := "PLCMemory".ProductBuffer.DelayTime, SystemTime := "PLCMemory".SystemTime, TriggerFeedback := "Move2Done".Q, TriggerMovement => "PLCMemory".ProductBuffer.MoveTrigger, InsertIndex => "PLCMemory".ProductBuffer.InsertIndex, ProductCount => "PLCMemory".ProductBuffer.ProductsCount, SystemTicks =>)
   END_RUNG
   // the same network as SCL:
   IF "Systeem RUN" AND #ActivateProductBufferV2 THEN
       "ProductBuffer_V2_DB"(SensorInput := "Sensor Op Band",   // "ProductBuffer_V2"
                             SensorManual := "PositionManagement".Demo_Pos.ManualSensorOverride,
                             TimeDelay := "PLCMemory".ProductBuffer.DelayTime,
                             SystemTime := "PLCMemory".SystemTime,
                             TriggerFeedback := "Move2Done".Q,
                             TriggerMovement => "PLCMemory".ProductBuffer.MoveTrigger,
                             InsertIndex => "PLCMemory".ProductBuffer.InsertIndex,
                             ProductCount => "PLCMemory".ProductBuffer.ProductsCount);
   END_IF;
END_REGION

REGION Network 31: ProductBuffer V3 - Currently in production testing)
   // This is the newest version of the Product Buffer, it's working great, and uses the encoder position of Axis 1 to ensure precise product place data. 
   // Switching between PB V2 and V3 can be done in the Automatiek Settings in the HMI, or manual trough tag M222.1
   RUNG wire#powerrail
      Contact( "Systeem RUN" )
      I_Contact( "ActivateProductBufferV3" )
      "ProductBuffer_V3_DB"(SensorInput := "Sensor Op Band", DevSensorInput := "PLCMemory".SimulateSensor, EncoderPosition := "Enc2", TriggerDistance := "PLCMemory".TriggerDistanceBand, TriggerFeedback := "Move2Done".Q, DirectionSign := -1, TriggerMovement => "PLCMemory".ProductBuffer_1.MoveTrigger, ProductCount => "PLCMemory".ProductBuffer_1.ProductsCount)
      Coil( "ProgramDebugger".ProgramDebugger1.Prog1_Dev_Steps[6].Enable )
   END_RUNG
   // the same network as SCL:
   "ProductBuffer_V3_DB"(EN := "Systeem RUN" AND NOT "ActivateProductBufferV3",   // "ProductBuffer_V3"
                         SensorInput := "Sensor Op Band",
                         DevSensorInput := "PLCMemory".SimulateSensor,
                         EncoderPosition := "Enc2",
                         TriggerDistance := "PLCMemory".TriggerDistanceBand,
                         TriggerFeedback := "Move2Done".Q,
                         DirectionSign := -1,
                         TriggerMovement => "PLCMemory".ProductBuffer_1.MoveTrigger,
                         ProductCount => "PLCMemory".ProductBuffer_1.ProductsCount,
                         ENO => #_w1);
   "ProgramDebugger".ProgramDebugger1.Prog1_Dev_Steps[6].Enable := #_w1;
END_REGION

REGION Network 32: Speed Select 25%
   // This Program ensures that when the machine is not in automatic mode, and the axis will always go to an safe position it will be done with a safe speed (25%)
   RUNG wire#powerrail
      I_Contact( "Systeem RUN" )
      { S7_GenerateENO := "TRUE" } Move(in := 50, out1 => "PositionManagement"."Axis 3".Values.Axis_Speed)
   END_RUNG
   // the same network as SCL:
   IF NOT "Systeem RUN" THEN "PositionManagement"."Axis 3".Values.Axis_Speed := 50; END_IF;
END_REGION

REGION Network 33: Speed Select 75%
   // This program ensures that when the machine is in automatic mode, the speed will rise up to 75% what is 105-110 Hz on the Frequency Converter.
   RUNG wire#powerrail
      Contact( "Systeem RUN" )
      { S7_GenerateENO := "TRUE" } Move(in := 75, out1 => "PositionManagement"."Axis 3".Values.Axis_Speed)
   END_RUNG
   // the same network as SCL:
   IF "Systeem RUN" THEN "PositionManagement"."Axis 3".Values.Axis_Speed := 75; END_IF;
END_REGION

REGION Network 34: Encoder Band Function Block
   // This Function Block is for controlling and reading encoder data from the Axis 1 SIKO IG09 encoder. More can be found on the wiki.
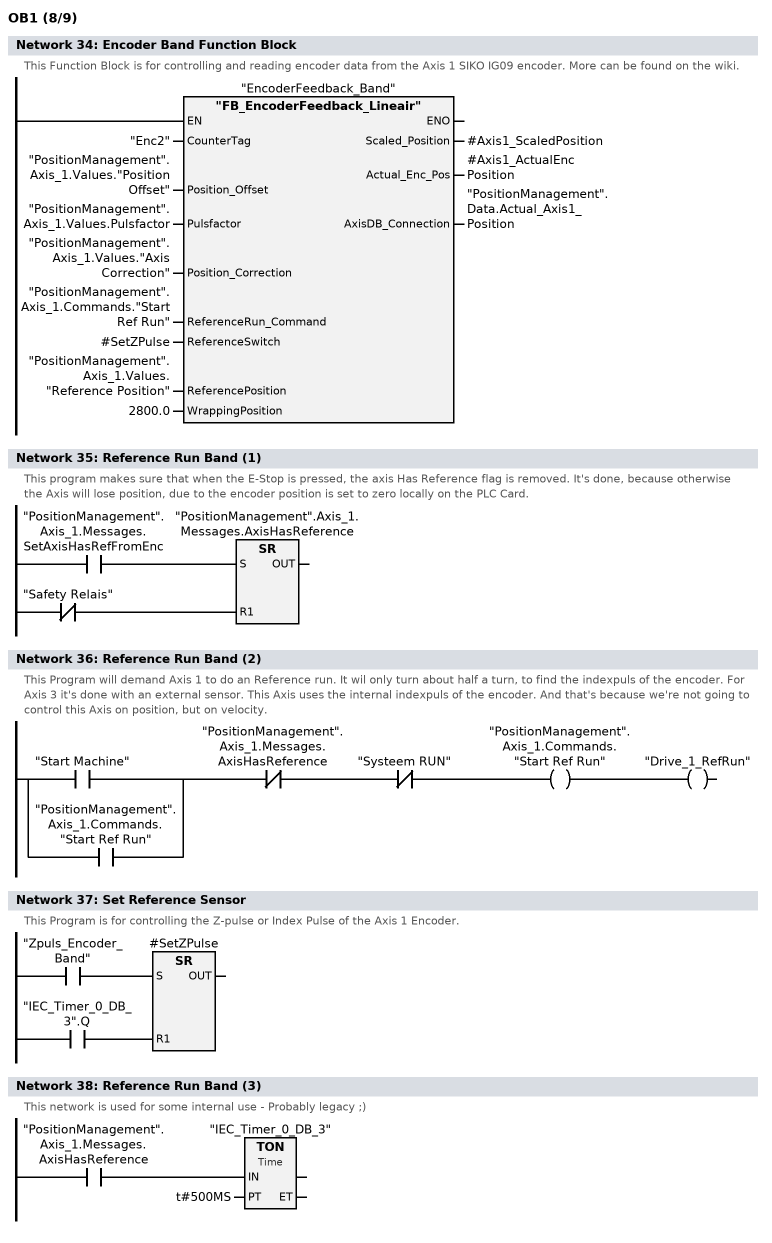
   RUNG wire#powerrail
      "EncoderFeedback_Band"(CounterTag := "Enc2", Position_Offset := "PositionManagement".Axis_1.Values."Position Offset", Pulsfactor := "PositionManagement".Axis_1.Values.Pulsfactor, Position_Correction := "PositionManagement".Axis_1.Values."Axis Correction", ReferenceRun_Command := "PositionManagement".Axis_1.Commands."Start Ref Run", ReferenceSwitch := #SetZPulse, ReferencePosition := "PositionManagement".Axis_1.Values."Reference Position", WrappingPosition := 2800.0, Scaled_Position => #Axis1_ScaledPosition, Actual_Enc_Pos => #Axis1_ActualEncPosition, AxisDB_Connection => "PositionManagement".Data.Actual_Axis1_Position)
   END_RUNG
   // the same network as SCL:
   "EncoderFeedback_Band"(CounterTag := "Enc2",   // "FB_EncoderFeedback_Lineair"
                          Position_Offset := "PositionManagement".Axis_1.Values."Position Offset",
                          Pulsfactor := "PositionManagement".Axis_1.Values.Pulsfactor,
                          Position_Correction := "PositionManagement".Axis_1.Values."Axis Correction",
                          ReferenceRun_Command := "PositionManagement".Axis_1.Commands."Start Ref Run",
                          ReferenceSwitch := #SetZPulse,
                          ReferencePosition := "PositionManagement".Axis_1.Values."Reference Position",
                          WrappingPosition := 2800.0,
                          Scaled_Position => #Axis1_ScaledPosition,
                          Actual_Enc_Pos => #Axis1_ActualEncPosition,
                          AxisDB_Connection => "PositionManagement".Data.Actual_Axis1_Position);
END_REGION

REGION Network 35: Reference Run Band (1)
   // This program makes sure that when the E-Stop is pressed, the axis Has Reference flag is removed. It's done, because otherwise the Axis will lose position, due to the encoder position is set to zero locally on the PLC Card.
   RUNG wire#powerrail
      Contact( "PositionManagement".Axis_1.Messages.SetAxisHasRefFromEnc )
      S_SR(operand := "PositionManagement".Axis_1.Messages.AxisHasReference, r1 := wire#w1)
   END_RUNG
   RUNG wire#powerrail
      I_Contact( "Safety Relais" )
   END_RUNG wire#w1
   // the same network as SCL:
   IF "PositionManagement".Axis_1.Messages.SetAxisHasRefFromEnc THEN
       "PositionManagement".Axis_1.Messages.AxisHasReference := TRUE;   // SR flip-flop
   END_IF;
   IF NOT "Safety Relais" THEN "PositionManagement".Axis_1.Messages.AxisHasReference := FALSE; END_IF;
END_REGION

REGION Network 36: Reference Run Band (2)
   // This Program will demand Axis 1 to do an Reference run. It wil only turn about half a turn, to find the indexpuls of the encoder. For Axis 3 it's done with an external sensor. This Axis uses the internal indexpuls of the encoder. And that's because we're not going to control this Axis on position, but on velocity.
   RUNG wire#powerrail
      Contact( "Start Machine" )
      wire#w1
      I_Contact( "PositionManagement".Axis_1.Messages.AxisHasReference )
      I_Contact( "Systeem RUN" )
      Coil( "PositionManagement".Axis_1.Commands."Start Ref Run" )
      Coil( "Drive_1_RefRun" )
   END_RUNG
   RUNG wire#powerrail
      Contact( "PositionManagement".Axis_1.Commands."Start Ref Run" )
   END_RUNG wire#w1
   // the same network as SCL:
   "PositionManagement".Axis_1.Commands."Start Ref Run" := ("Start Machine" OR "PositionManagement".Axis_1.Commands."Start Ref Run") AND NOT "PositionManagement".Axis_1.Messages.AxisHasReference AND NOT "Systeem RUN";
   "Drive_1_RefRun" := "PositionManagement".Axis_1.Commands."Start Ref Run";
END_REGION

REGION Network 37: Set Reference Sensor
   // This Program is for controlling the Z-pulse or Index Pulse of the Axis 1 Encoder.
   RUNG wire#powerrail
      Contact( "Zpuls_Encoder_Band" )
      S_SR(operand := #SetZPulse, r1 := wire#w1)
   END_RUNG
   RUNG wire#powerrail
      Contact( "IEC_Timer_0_DB_3".Q )
   END_RUNG wire#w1
   // the same network as SCL:
   IF "Zpuls_Encoder_Band" THEN
       #SetZPulse := TRUE;   // SR flip-flop
   END_IF;
   IF "IEC_Timer_0_DB_3".Q THEN #SetZPulse := FALSE; END_IF;
END_REGION

REGION Network 38: Reference Run Band (3)
   // This network is used for some internal use - Probably legacy ;)
   RUNG wire#powerrail
      Contact( "PositionManagement".Axis_1.Messages.AxisHasReference )
      { S7_Templates := "time_type := Time" } "IEC_Timer_0_DB_3".TON(pt := t#500MS, et =>)
   END_RUNG
   // the same network as SCL:
   "IEC_Timer_0_DB_3".TON(IN := "PositionManagement".Axis_1.Messages.AxisHasReference, PT := t#500MS);
END_REGION

REGION Network 39: SystemTime
   // This network will read the PLC Uptime. It was used for timestamp purposes.
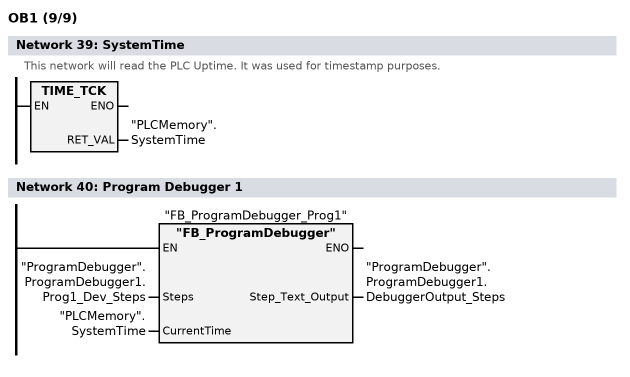
   RUNG wire#powerrail
      TIME_TCK(RET_VAL => "PLCMemory".SystemTime)
   END_RUNG
   // the same network as SCL:
   "PLCMemory".SystemTime := TIME_TCK();
END_REGION

REGION Network 40: Program Debugger 1
   RUNG wire#powerrail
      "FB_ProgramDebugger_Prog1"(Steps := "ProgramDebugger".ProgramDebugger1.Prog1_Dev_Steps, CurrentTime := "PLCMemory".SystemTime, Step_Text_Output => "ProgramDebugger".ProgramDebugger1.DebuggerOutput_Steps)
   END_RUNG
   // the same network as SCL:
   "FB_ProgramDebugger_Prog1"(Steps := "ProgramDebugger".ProgramDebugger1.Prog1_Dev_Steps,   // "FB_ProgramDebugger"
                           CurrentTime := "PLCMemory".SystemTime,
                           Step_Text_Output => "ProgramDebugger".ProgramDebugger1.DebuggerOutput_Steps);
END_REGION
END_ORGANIZATION_BLOCK
